// TIA Portal V17 export
// export: Created 2022-07-20T06:59:48.4198379Z, ExportSetting WithDefaults, DisplayName Totally Integrated Automation Portal, DisplayVersion V17, DisplayName TIA Portal Openness, DisplayVersion V17, DisplayName TIA Portal Version Control Interface, DisplayVersion V17, DisplayName SINAMICS Startdrive Advanced, DisplayVersion V17, DisplayName SINAMICS Startdrive G130, G150, S120, S150, SINAMICS MV, S210, DisplayVersion V17, DisplayName SINAMICS Startdrive G110M, G120, G120C, G120D, G120P, G115D, DisplayVersion V17, DisplayName STEP 7 Professional, DisplayVersion V17, DisplayName STEP 7 Safety, DisplayVersion V17, DisplayName WinCC Advanced, DisplayVersion V17
FUNCTION_BLOCK "FB10200_ModuleKindOfAlarmManagement"   // FB10200, LAD
{ S7_Optimized_Access := 'TRUE' }
VERSION : 0.1
// stored: AutoNumber false, IsIECCheckEnabled false, IsRetainMemResEnabled false, MemoryReserve 100, SetENOAutomatically false, UDAEnableTagReadback false
   VAR_INPUT
      FirstStartDetected : Bool;
      NormalStopDetected : Bool;
      QuickStopDetected : Bool;
      ResetMemory : Bool;
      Bypass : Bool;
   END_VAR
   VAR_OUTPUT
      FirstStartMemory : Bool;
      NormalStopMemory : Bool;
      QuickStopMemory : Bool;
   END_VAR
   VAR
      R_TRIG_FirstStartDetected : R_TRIG;
      R_TRIG_NormalStopDetected { S7_SetPoint := 'True'} : R_TRIG;
      R_TRIG_QuickStopDetected { S7_SetPoint := 'True'} : R_TRIG;
      R_TRIG_ResetMemory { S7_SetPoint := 'True'} : R_TRIG;
   END_VAR
BEGIN

REGION Network 1 (SCL): Edge Signals & Timers
   REGION EDGE SIGNALS
       #R_TRIG_FirstStartDetected(CLK := #FirstStartDetected);
       #R_TRIG_NormalStopDetected(CLK := #NormalStopDetected);
       #R_TRIG_QuickStopDetected(CLK := #QuickStopDetected);
       #R_TRIG_ResetMemory(CLK := #ResetMemory);
   END_REGION
END_REGION

REGION Network 2 (SCL): Memory Management
   IF NOT(#Bypass) THEN
       IF #R_TRIG_FirstStartDetected.Q THEN
           #FirstStartMemory := TRUE;
           #NormalStopMemory := FALSE;
           #QuickStopMemory := FALSE;
       ELSIF #R_TRIG_NormalStopDetected.Q THEN
           #FirstStartMemory := FALSE;
           #NormalStopMemory := TRUE;
           #QuickStopMemory := FALSE;
       ELSIF #R_TRIG_QuickStopDetected.Q THEN
           #FirstStartMemory := FALSE;
           #NormalStopMemory := FALSE;
           #QuickStopMemory := TRUE;
       ELSIF #R_TRIG_ResetMemory.Q THEN
           #FirstStartMemory := FALSE;
           #NormalStopMemory := FALSE;
           #QuickStopMemory := FALSE;
       END_IF;
   ELSE
       #FirstStartMemory := FALSE;
       #NormalStopMemory := TRUE;
       #QuickStopMemory := FALSE;
   END_IF;
END_REGION
END_FUNCTION_BLOCK
